// TIA Portal project "Project_Setting" (V18)

(* hardware
DEVICE "S7-1500/ET200MP station_1"  S7-1500 station
   slot 0: "PM 190W 120/230VAC"  PM 190W 120/230VAC  6EP1333-4BA00
   slot 0: "Rail_0"  Rack  6ES7 590-1***0-0AA0
   slot 1: "PLC_1"  CPU 1516-3 PN/DP  6ES7 516-3AN01-0AB0  V2.0
      slot 3: "CPU display_1"  6ES7591-1BA00-0AA0
      slot 32768: "PROFINET interface_1"  X1
         slot 32769: "Port_1"  X1 P1
         slot 32770: "Port_2"  X1 P2
      slot 33024: "PROFINET interface_2"  X2
         slot 33025: "Port_1"  X2 P1
      slot 33280: "DP interface_1"  X3
   slot 2: "DI 32x24VDC HF_1"  DI 32x24VDC HF  6ES7 521-1BL00-0AB0  V2.2
   slot 3: "DQ 32x24VDC/0.5A HF_1"  DQ 32x24VDC/0.5A HF  6ES7 522-1BL01-0AB0  V1.1
   slot 4: "AI 8xU/I/RTD/TC ST_1"  AI 8xU/I/RTD/TC ST  6ES7 531-7KF00-0AB0  V2.2
   slot 5: "AQ 4xU/I HF_1"  AQ 4xU/I HF  6ES7 532-5ND00-0AB0  V1.1
*)

// ===== PLC "PLC_1"  CPU 1516-3 PN/DP =====

VAR_GLOBAL   // PLC tag table "Default tag table"
   "IN_00" AT %I0.7 : Bool;
   "IN_01" AT %I0.1 : Bool;
   "IN_02" AT %I0.2 : Bool;
   "OUT_00" AT %Q0.0 : Bool;
   "OUT_01" AT %Q0.1 : Bool;
   "OUT_02" AT %Q0.2 : Bool;
   "Tag_1" AT %I0.0 : Bool;
   "Tag_2" AT %I0.3 : Bool;
   "Tag_3" AT %Q0.3 : Bool;
END_VAR

VAR_GLOBAL CONSTANT   // PLC tag table "Default tag table"
   "Max_Time" : Time := T#2000MS;   // 타이머 최대 시간 설정값 상수
END_VAR

DATA_BLOCK "SELF_HOLDING_FB01_DB"   // DB3
{ S7_Optimized_Access := 'TRUE' }
VERSION : 0.1
// stored: InstanceOfName SELF_HOLDING_FB01
"SELF_HOLDING_FB01"
BEGIN
END_DATA_BLOCK

// folder: System blocks/Program resources

DATA_BLOCK "IEC_Timer_0_DB"   // DB1
{ S7_Optimized_Access := 'TRUE' }
AUTHOR : Simatic
FAMILY : IEC
NAME : IEC_TMR
VERSION : 1.0
// stored: InstanceOfName IEC_TIMER
"IEC_TIMER"
BEGIN
END_DATA_BLOCK

DATA_BLOCK "IEC_Timer_0_DB_1"   // DB2
{ S7_Optimized_Access := 'TRUE' }
AUTHOR : Simatic
FAMILY : IEC
NAME : IEC_TMR
VERSION : 1.0
// stored: InstanceOfName IEC_TIMER
"IEC_TIMER"
BEGIN
END_DATA_BLOCK

// folder: (top level)

FUNCTION_BLOCK "SELF_HOLDING_FB01"   // FB1, LAD
{ S7_Optimized_Access := 'TRUE' }
VERSION : 0.1
   VAR_INPUT
      SET : Bool;
      RST : Bool;
   END_VAR
   VAR_OUTPUT
      OUT : Bool;
   END_VAR
   VAR
      K1 : Bool;
   END_VAR
BEGIN

REGION Network 1
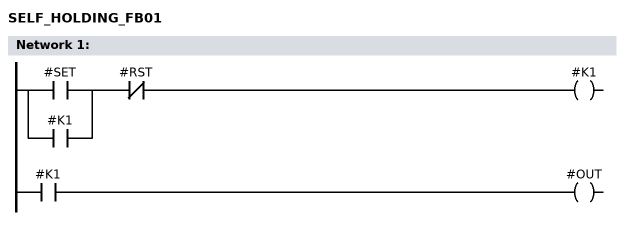
   RUNG wire#powerrail
      Contact( #SET )
      wire#w1
      I_Contact( #RST )
      Coil( #K1 )
   END_RUNG
   RUNG wire#powerrail
      Contact( #K1 )
   END_RUNG wire#w1
   RUNG wire#powerrail
      Contact( #K1 )
      Coil( #OUT )
   END_RUNG
   // the same network as SCL:
   #K1 := (#SET OR #K1) AND NOT #RST;
   #OUT := #K1;
END_REGION
END_FUNCTION_BLOCK

ORGANIZATION_BLOCK "Main"   // OB1, LAD, ProgramCycle
TITLE = "Main Program Sweep (Cycle)"
{ S7_Optimized_Access := 'TRUE' }
VERSION : 0.1
   VAR_INPUT
      Initial_Call : Bool;   // Initial call of this OB
      Remanence : Bool;   // =True, if remanent data are available
   END_VAR
BEGIN

REGION Network 1
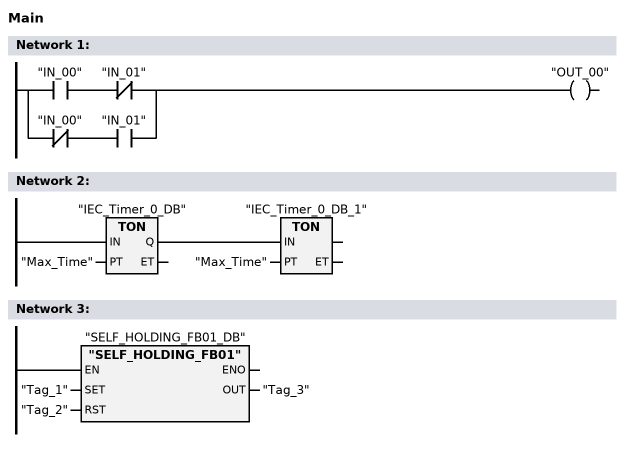
   RUNG wire#powerrail
      Contact( "IN_00" )
      I_Contact( "IN_01" )
      wire#w1
      Coil( "OUT_00" )
   END_RUNG
   RUNG wire#powerrail
      I_Contact( "IN_00" )
      Contact( "IN_01" )
   END_RUNG wire#w1
   // the same network as SCL:
   "OUT_00" := ("IN_00" AND NOT "IN_01") OR (NOT "IN_00" AND "IN_01");
END_REGION

REGION Network 2
   "IEC_Timer_0_DB".TON(IN := TRUE, PT := "Max_Time");
   "IEC_Timer_0_DB_1".TON(IN := "IEC_Timer_0_DB".Q, PT := "Max_Time");
END_REGION

REGION Network 3
   RUNG wire#powerrail
      "SELF_HOLDING_FB01_DB"(SET := "Tag_1", RST := "Tag_2", OUT => "Tag_3")
   END_RUNG
   // the same network as SCL:
   "SELF_HOLDING_FB01_DB"(SET := "Tag_1", RST := "Tag_2", OUT => "Tag_3");   // "SELF_HOLDING_FB01"
END_REGION
END_ORGANIZATION_BLOCK